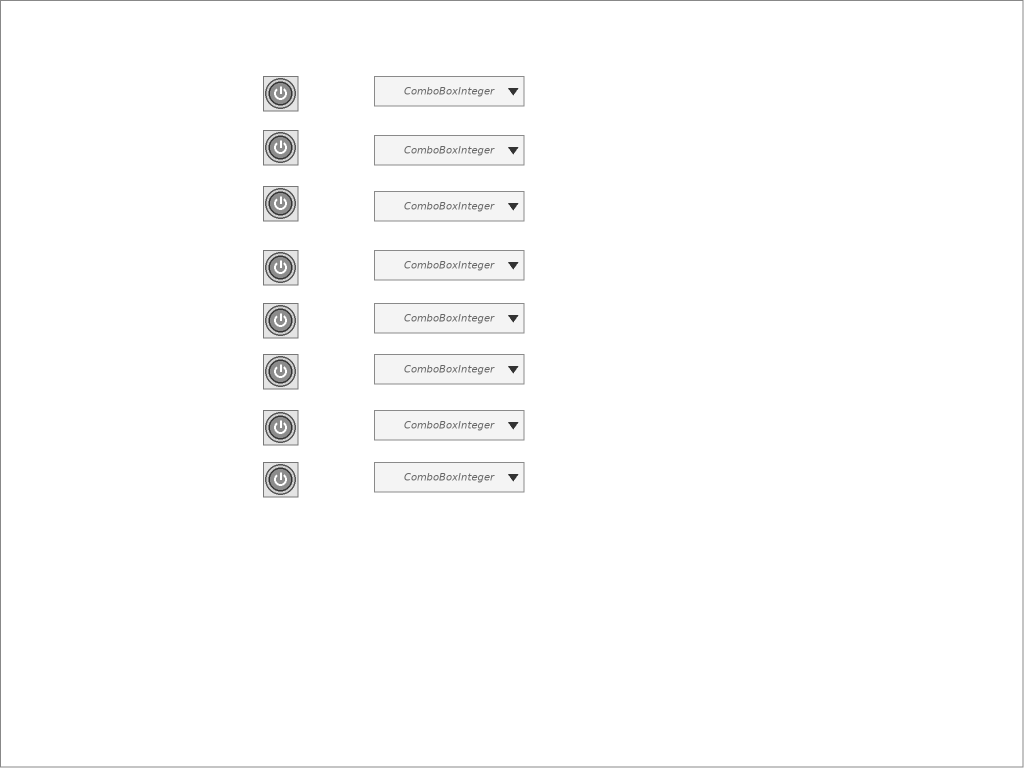
VISUALIZATION Visualization  // 1024x768
    ComboBoxInteger (374,76 150x30), variable: MAIN.outRefs.out1, text list: 'tl_OutputNames'
    ComboBoxInteger (374,135 150x30), variable: MAIN.outRefs.out2, text list: 'tl_OutputNames'
    ComboBoxInteger (374,191 150x30), variable: MAIN.outRefs.out3, text list: 'tl_OutputNames'
    ComboBoxInteger (374,250 150x30), variable: MAIN.outRefs.out4, text list: 'tl_OutputNames'
    ComboBoxInteger (374,303 150x30), variable: MAIN.outRefs.out5, text list: 'tl_OutputNames'
    ComboBoxInteger (374,354 150x30), variable: MAIN.outRefs.out6, text list: 'tl_OutputNames'
    ComboBoxInteger (374,410 150x30), variable: MAIN.outRefs.out7, text list: 'tl_OutputNames'
    ComboBoxInteger (374,462 150x30), variable: MAIN.outRefs.out8, text list: 'tl_OutputNames'
    PowerSwitch (263,76 35x35), variable: MAIN.outs[1], behaviour: TAP, style: Switch-PowerSwitch-Gray
    PowerSwitch (263,130 35x35), variable: MAIN.outs[2], behaviour: TAP, style: Switch-PowerSwitch-Gray
    PowerSwitch (263,186 35x35), variable: MAIN.outs[3], behaviour: TAP, style: Switch-PowerSwitch-Gray
    PowerSwitch (263,250 35x35), variable: MAIN.outs[4], behaviour: TAP, style: Switch-PowerSwitch-Gray
    PowerSwitch (263,303 35x35), variable: MAIN.outs[5], behaviour: TAP, style: Switch-PowerSwitch-Gray
    PowerSwitch (263,354 35x35), variable: MAIN.outs[6], behaviour: TAP, style: Switch-PowerSwitch-Gray
    PowerSwitch (263,410 35x35), variable: MAIN.outs[7], behaviour: TAP, style: Switch-PowerSwitch-Gray
    PowerSwitch (263,462 35x35), variable: MAIN.outs[8], behaviour: TAP, style: Switch-PowerSwitch-Gray
END_VISUALIZATION

(* stored: Version 1.1.0.1
   Visu Visualization: Id {4e31ec56-56cd-4824-9d0e-640e2bba57e8} *)
